(* PLC project Unknown, Unknown Unknown 1 *)
(* stored: creationDateTime 2024-06-18T10:21:19.081890Z, language english *)

PROGRAM pou1
  VAR  (* added by the conversion: wires and edge detectors of the diagram *)
    _AND3_OUT : BOOL;
    _AND2_OUT : BOOL;
    _AND7_OUT : BOOL;
    _AND1_OUT : BOOL;
    _AND4_OUT : BOOL;
    _AND8_OUT : BOOL;
    _AND6_OUT : BOOL;
    _AND0_OUT : BOOL;
    _AND5_OUT : BOOL;
  END_VAR

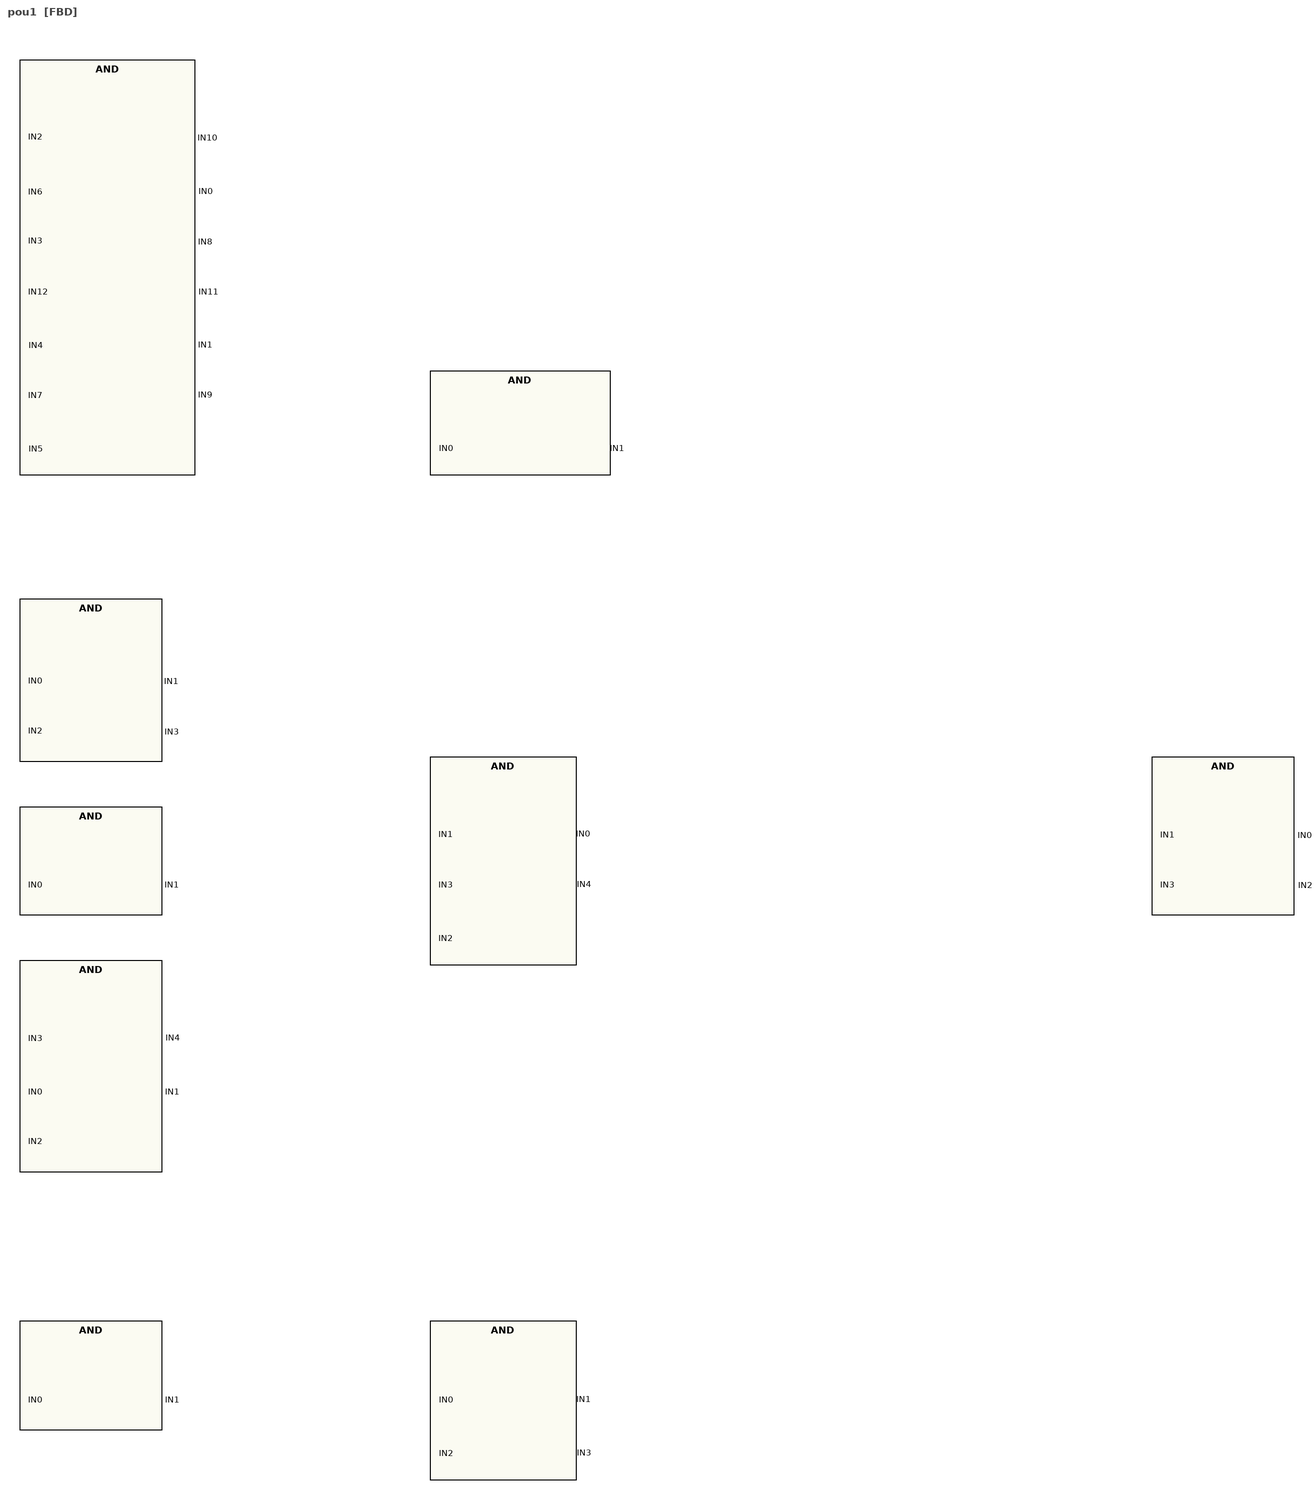
(* FBD diagram, written out as Structured Text *)
_AND3_OUT := AND();
_AND2_OUT := AND();
_AND7_OUT := AND();
_AND1_OUT := AND();
_AND4_OUT := AND();
_AND8_OUT := AND();
_AND6_OUT := AND();
_AND0_OUT := AND();
_AND5_OUT := AND();
END_PROGRAM
